Fanuc KAREL source: kb00107.KL

-- PROVISIONAL review KL for V770-1; original PC SHA256 59e7865d22c73e1dddc8f2c5d5113b3c4d649a1d989b7b1a1212d30b8564b568
-- Incomplete behavior may be omitted. Consult companion uncertainty JSON. Do not deploy.
PROGRAM KB00107
%NOLOCKGROUP
VAR
  RESULT : BOOLEAN
-- UNRESOLVED_DECL P1 type=000106
BEGIN
  -- UNRESOLVED_PC offsets 5-28; opcodes 27,22,1C,27,9D,76,23
  -- UNRESOLVED_PC offsets 33-37; opcodes 7F
END KB00107
